PROGRAM SERIALCOMMS
VAR
END_VAR

GVL.fbSpindle.M_SerialLineControl();

END_PROGRAM

(* stored: Version 1.1.0.1, ProductVersion 3.1.4024.9
   POU SERIALCOMMS: Id {bde08e60-56d8-42a4-bd78-c5daeeb46c51}, SpecialFunc None *)
